TEXTLIST TextList_RTRstate
  0 = 'off'
  1 = 'initializing'
  2 = 'ready'
  4 = 'active'
  5 = 'tensioning'
  6 = 'Tensioned_locked'
  8 = 'tensioned'
  9 = 'untensioning'
  10 = 'setting_off'
  13 = 'brake_enabled'
  100 = 'error'
   = ''
END_TEXTLIST

(* stored: Version 1.1.0.1, ProductVersion 3.1.4024.11
   TextList TextList_RTRstate: Id {5c4bf2b9-8f39-4763-97c6-45d9bcacfb5d} *)
